PROGRAM P03_DiskSize
VAR
	fbSize						:FB_PythonScript;
	bReadAfterPowerUp			:BOOL;
	tonReadAfterPowerUpDelay	:TON;
END_VAR

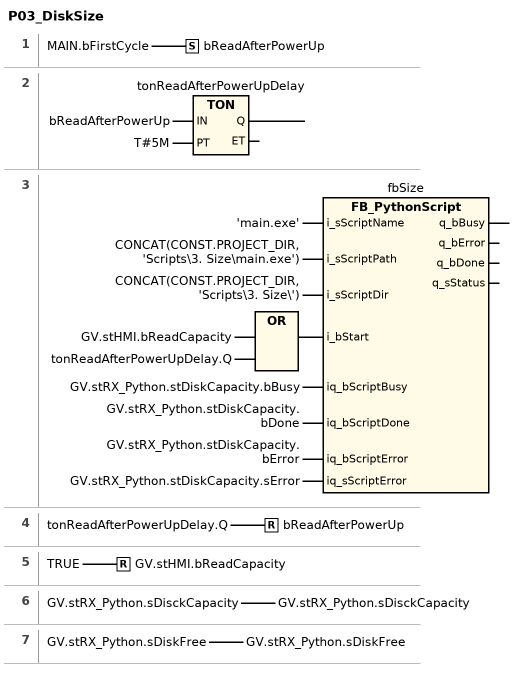
// NETWORK 1
bReadAfterPowerUp S= MAIN.bFirstCycle;

// NETWORK 2
tonReadAfterPowerUpDelay(IN := bReadAfterPowerUp, PT := T#5M); // TON

// NETWORK 3
fbSize(
    i_sScriptName := 'main.exe',
    i_sScriptPath := CONCAT(CONST.PROJECT_DIR,'Scripts\3. Size\main.exe'),
    i_sScriptDir := CONCAT(CONST.PROJECT_DIR,'Scripts\3. Size\'),
    i_bStart := GV.stHMI.bReadCapacity OR tonReadAfterPowerUpDelay.Q,
    iq_bScriptBusy := GV.stRX_Python.stDiskCapacity.bBusy,
    iq_bScriptDone := GV.stRX_Python.stDiskCapacity.bDone,
    iq_bScriptError := GV.stRX_Python.stDiskCapacity.bError,
    iq_sScriptError := GV.stRX_Python.stDiskCapacity.sError); // FB_PythonScript

// NETWORK 4
bReadAfterPowerUp R= tonReadAfterPowerUpDelay.Q;

// NETWORK 5
GV.stHMI.bReadCapacity R= TRUE;

// NETWORK 6
GV.stRX_Python.sDisckCapacity := GV.stRX_Python.sDisckCapacity;

// NETWORK 7
GV.stRX_Python.sDiskFree := GV.stRX_Python.sDiskFree;

END_PROGRAM

(* stored: Version 1.1.0.1, ProductVersion 3.1.4026.13
   POU P03_DiskSize: Id {37c73627-27c3-4fae-9810-f82ba81eb48e}, SpecialFunc None *)
